(* PLC project  *)

PROGRAM MAIN
  VAR_INPUT
    start : BOOL;
  END_VAR

          
          start := TRUE;
          
        
END_PROGRAM
